(* Logix 5000 project; controller GitHubTest 1756-L72 rev 20.11; software revision 20.05 *)

TASK MainTask (continuous, watchdog 500 ms) : MainProgram

MODULES
   Local : 1756-L72 (ICP 0, rev 20.11)
END_MODULES

VAR_GLOBAL   (* controller tags *)
   Output1 : BOOL;
   Output2 : BOOL;
   Output3 : BOOL;
   ST_OUT : BOOL;
   ST_OUT2 : BOOL;
   Variable1 : BOOL;
   Variable2 : BOOL;
   Variable3 : BOOL;
END_VAR

PROGRAM MainProgram   (* main routine MainRoutine *)

ROUTINE MainRoutine   (* ladder *)
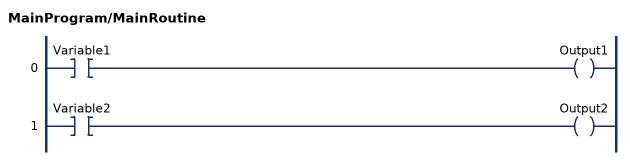
   0: XIC(Variable1)OTE(Output1);
   1: XIC(Variable2)OTE(Output2);
END_ROUTINE

ROUTINE ST_Test   (* structured text *)
   if Output1 and Output2 then
    ST_OUT := 1;
   end_if;
   
END_ROUTINE
END_PROGRAM
